FUNCTION_BLOCK FB_LinearEquation
VAR_INPUT
	x1: REAL;
	y1: REAL;
	x2: REAL;
	y2: REAL;
	x: REAL;
END_VAR
VAR_OUTPUT
	y: REAL;
END_VAR
VAR
	a: REAL;
	b: REAL;
END_VAR

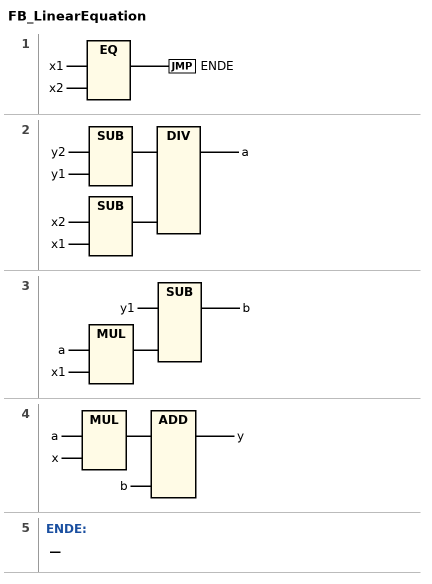
// NETWORK 1
IF x1 = x2 THEN JMP ENDE; END_IF

// NETWORK 2
a := (y2 - y1) / (x2 - x1);

// NETWORK 3
b := y1 - a * x1;

// NETWORK 4
y := a * x + b;

// NETWORK 5
ENDE: ;

END_FUNCTION_BLOCK

(* stored: Version 1.1.0.1, ProductVersion 3.1.4024.12
   POU FB_LinearEquation: Id {5d3ade1f-b61e-41c2-837f-c9e37e220235}, SpecialFunc None *)
